PROGRAM GeneralPlc
VAR
END_VAR
(* End *)

(* General *)

(* Analog input to output *)
	nAnalogOutP10 := nAnalogInR10;
	
(* Led on/off *)
	bLedH25 := bSwitchS25;

(* End *)

END_PROGRAM

(* stored: Version 1.1.0.1, ProductVersion 3.1.4020.3
   POU GeneralPlc: Id {40442ba5-5468-42d6-b755-fa74013c25b0}, SpecialFunc None *)
